FUNCTION_BLOCK FB_SimuMoverAxis
VAR_INPUT
    xIN_StopMover : BOOL; // stop the mover from movinf
END_VAR
VAR_OUTPUT
    outSimuCurrentPos : Pos2D_t; // Mover position, expressed as slot number
    outSimuCurrentRot : INT;     // mover current rotation
    isInPos           : BOOL;    // true when targetPos = currentPos
END_VAR
VAR
    // with tick rate at 10ms, a value of 10 gives us 1m/s
    _Velocity    : LREAL := 0;     // Mover velocity, expressed as mm per tick, max is 10m/s
    _ErrorState  : INT   := 0;     // error state, not used
    _TargetPos   : LREAL := 0;     // last target pos
    _CurrentPos  : LREAL := 0;     // Current Pos, but with more resolution than the pixel
    _IsColliding : BOOL  := FALSE; // When true, the mover should not move
    _LastPos     : LREAL := 0;     // last position, used to trigger the xStuck flag
    _xStuck      : BOOL;           // true when the axis does not move
    _willCollide : BOOL := FALSE;  // TRUE if a collision will occure with the current velocity

    {attribute 'hide'}
    _lrNextStopPos : LREAL; // local variable used to get next stop

    _iID : INT := 0; // instance ID, is set during FB_Init using the value of _iInstanceCounter 
	
	_CurrentDir : MoverDirection_e := MoverDirection_e.Farward;
END_VAR

VAR_TEMP
	_MoverAccel : LREAL;	// Mover acceleration, can be positive or negative depending on the direction
END_VAR

VAR CONSTANT
    MAX_POS            : LREAL := CONST.MAX_TRACK_LENGTH; // should be defined elsewhere ...
    MAX_SIZE           : LREAL := CONST.MAX_MOVER_SIZE;   // Maxium size of the mover
    //MOVER_ACCEL        : LREAL := 0.1;                      // Mover acceleration, in mm/tick^2
    //MOVER_VELOCITY_MAX : LREAL := 20;                     // Mover velocity, expressed as mm per tick, max is 10m/s
    MOVER_VELOCITY_MIN : LREAL := 1;                      // Mover velocity, expressed as mm per tick, max is 10m/s
END_VAR
VAR_STAT
    _iInstanceCounter : INT := 1; // instance counter
END_VAR

IF NOT xIN_StopMover THEN // Do not change momemtum when we stop the movers from HMI
    IF MoverDirection_e.Farward = THIS^._CurrentDir THEN
        _MoverAccel := SIMU.lrAccelMover;
    ELSE
        _MoverAccel := -SIMU.lrAccelMover;
    END_IF

    IF NOT _IsColliding THEN

        IF THIS^.GetStopLen(_Velocity, SIMU.lrAccelMover) >= DistToTravel(_CurrentPos, _TargetPos) OR
           THIS^._willCollide THEN
            _Velocity := _Velocity - _MoverAccel;

        ELSIF SIMU.lrSpeedMover > ABS(_Velocity) AND _CurrentPos <> _TargetPos THEN
            _Velocity := _Velocity + _MoverAccel;

        END_IF
    ELSE
        _Velocity := _Velocity - _MoverAccel;
    END_IF
END_IF

// protect max and min speed
IF SIMU.lrSpeedMover < ABS(_Velocity) THEN
    IF MoverDirection_e.Farward = THIS^._CurrentDir THEN
        _Velocity := SIMU.lrSpeedMover;
    ELSE
        _Velocity := -SIMU.lrSpeedMover;
    END_IF
ELSIF ABS(_Velocity) < MOVER_VELOCITY_MIN THEN
    IF MoverDirection_e.Farward = THIS^._CurrentDir THEN
        _Velocity := MOVER_VELOCITY_MIN;
    ELSE
        _Velocity := -MOVER_VELOCITY_MIN;
    END_IF
END_IF

IF NOT _IsColliding AND NOT xIN_StopMover THEN

    IF DistToTravel(_CurrentPos, _TargetPos) > ABS(_Velocity) THEN
        _CurrentPos := _CurrentPos + _Velocity;

    ELSE
        _CurrentPos := _TargetPos;
        _Velocity   := 0;

    END_IF
END_IF

IF _CurrentPos >= MAX_POS THEN
    _CurrentPos := _CurrentPos - MAX_POS;
    // we prevent the stuck flag to be true at the end of the track
    THIS^._LastPos := THIS^._LastPos - MAX_POS;
END_IF

isInPos := EqualDelta(_CurrentPos, _TargetPos, 1.0); // we use delta comparison beacause axis is always at a low value 
outSimuCurrentPos
    := THIS^.ResolvePos(this^.CurrentPos, outSimuCurrentRot);

_xStuck        := (THIS^._CurrentPos < (THIS^._LastPos + _Velocity)) AND NOT isInPos;
THIS^._LastPos := THIS^._CurrentPos;

PROPERTY CurrentPos : LREAL
GET
IF CONST.USE_SIMULATION THEN
    CurrentPos := _CurrentPos;
ELSE
    CurrentPos := TO_LREAL(gMoverAxis.I_BuR_MoverAxis.asStruct[THIS^._iID].diCurrentPos_um) / 1000.0;
END_IF
END_GET
SET
END_SET
END_PROPERTY

PROPERTY CurrentVelocity : LREAL
GET
CurrentVelocity := THIS^._Velocity;
END_GET
SET
END_SET
END_PROPERTY

METHOD FB_init : BOOL
VAR_INPUT
    bInitRetains : BOOL; // if TRUE, the retain variables are initialized (warm start / cold start)
    bInCopyCode  : BOOL; // if TRUE, the instance afterwards gets moved into the copy code (online change)

    PosInit : LREAL; // initial position at startup
END_VAR
THIS^._iID := THIS^._iInstanceCounter;
THIS^._iInstanceCounter := THIS^._iInstanceCounter +1;
IF PosInit < THIS^.MAX_POS THEN
    THIS^._CurrentPos := PosInit;
ELSE
    THIS^._CurrentPos := 0;
END_IF
END_METHOD

METHOD PRIVATE GetStopLen : LREAL
VAR_INPUT
    currentVelocity : LREAL;
    currentAccel    : LREAL;
END_VAR
VAR
    tickToStop : INT;
END_VAR
// This function search the position we will get if we stop now
//
// (velocity)
//     ^          _________   <- we are here, at the end of the top slope
//     |        /          \
//     |       /            \
//     |   ___/              \______
//     |     
//     ┼------------------------------>  (time)
//
// (position)
//     ^ 
//     |                      _________
//     |                  .../
//     |               ../    ^
//     |            ../       |
//     |          ../         we search this position
//     |   ___.../
//     | 
//     ┼------------------------------>  (time)

IF currentAccel <= 0 THEN
    ASSERT(currentAccel > 0);
    RETURN;
END_IF

// TO_INT floor the result, and we need at least 1 tick to stop
tickToStop := TO_INT(currentVelocity / currentAccel) + 1;

GetStopLen := tickToStop * currentVelocity / 2;
END_METHOD

// only check the collision in one way, this prevent
// all the mover chain to be stucked
METHOD IsColliding : BOOL
VAR_INPUT
    nextMover : REFERENCE TO FB_SimuMoverAxis;
END_VAR
IsColliding := FALSE;

IF DistToTravel(THIS^.CurrentPos, nextMover.CurrentPos) <= CONST.MAX_MOVER_SIZE THEN
    IsColliding := TRUE;

END_IF

THIS^._IsColliding := IsColliding;
END_METHOD

METHOD PUBLIC MoveTo : REFERENCE TO FB_SimuMoverAxis
VAR_INPUT
    Position : LREAL; // move the axis to this position
END_VAR
THIS^._TargetPos := Position;
THIS^._CurrentDir := MoverDirection_e.Farward;
isInPos := THIS^._CurrentPos = THIS^._TargetPos;
MoveTo REF= THIS^;
END_METHOD

// Move relatively of this position
// With this function, a negative value move the mover at the reverse direction
METHOD RelMoveTo : REFERENCE TO FB_SimuMoverAxis
VAR_INPUT
    RelativePos : LREAL; // move the axis to this amount¨
END_VAR
THIS^._TargetPos := THIS^._TargetPos + RelativePos;

IF RelativePos >= 0 THEN
    THIS^._CurrentDir := MoverDirection_e.Farward;
ELSE
    THIS^._CurrentDir := MoverDirection_e.Reverse;
END_IF

isInPos   := THIS^._CurrentPos = THIS^._TargetPos;
RelMoveTo REF= THIS^;
END_METHOD

METHOD ResolvePos : Pos2D_t
VAR_INPUT
    inX      : LREAL;
    rotation : REFERENCE TO INT;
END_VAR
VAR CONSTANT
    (* The track has this dimension in reality
              __________
     1000mm (___________) 1000 mm
              4000 mm
			  
     and we map it like that:
	   __   80 (radius)
	  |  |
	  |  |  800
	  |  |
	  |__|
	        80 (raidus)
    *)
    START_X     : DINT  := 0;
    START_Y     : DINT  := 0;
    MAX_SIMU_DX : DINT  := 120;
    MAX_SIMU_DY : DINT  := 800;
    RADIUS_X    : LREAL := 60.0;
    RADIUS_Y    : LREAL := 80.0;

    FIRST_RADIUS_START  : LREAL := 4000;
    FIRST_RADIUS_END    : LREAL := 5000;
    SECOND_RADIUS_START : LREAL := 9000;
    SECOND_RADIUS_END   : LREAL := 10000;
END_VAR

VAR
    x_rad_calc : LREAL;
    y_rad_calc : LREAL;
    FACTOR_Y   : LREAL;
END_VAR
FACTOR_Y := FIRST_RADIUS_START / MAX_SIMU_DY;

IF inX < 0 THEN
    ResolvePos.x := START_X;
    ResolvePos.y := START_Y;
    rotation     := 0;

ELSIF inX >= 0 AND inX <= FIRST_RADIUS_START THEN
    ResolvePos.x := START_X;
    ResolvePos.y := START_Y + TO_DINT(inX / FACTOR_Y);
    rotation     := 0;

ELSIF inX > FIRST_RADIUS_START AND inX < FIRST_RADIUS_END THEN

    // should go between -1RAD and +1RAD
    x_rad_calc   := ((inX - FIRST_RADIUS_START) * 2 / (FIRST_RADIUS_END - FIRST_RADIUS_START) - 1) * PI / 2;
    ResolvePos.x := TO_DINT(SIN(x_rad_calc) * RADIUS_X) + START_X + TO_DINT(RADIUS_X);

    // should go from 0RAD to 1RAD, then 0RAD
    y_rad_calc   := (1 - (inX - FIRST_RADIUS_START) * 2 / (FIRST_RADIUS_END - FIRST_RADIUS_START)) * PI / 2;
    ResolvePos.y := TO_DINT(COS(y_rad_calc) * RADIUS_Y + START_Y + MAX_SIMU_DY);

    rotation := TO_INT(SIN(x_rad_calc) * 90 + 90);

ELSIF inX >= FIRST_RADIUS_END AND inX <= SECOND_RADIUS_START THEN
    ResolvePos.x := START_X + MAX_SIMU_DX;
    ResolvePos.y := START_Y + MAX_SIMU_DY - TO_DINT((inX - FIRST_RADIUS_END) / FACTOR_Y);
    rotation     := 180;

ELSIF inX > SECOND_RADIUS_START AND inX < SECOND_RADIUS_END THEN
    // should go between -1RAD and +1RAD
    x_rad_calc   := ((inX - SECOND_RADIUS_START) * 2 / (SECOND_RADIUS_END - SECOND_RADIUS_START) - 1) * PI / 2;
    ResolvePos.x := START_X - TO_DINT(SIN(x_rad_calc) * RADIUS_X) + TO_DINT(RADIUS_X);

    // should go from 0RAD to 1RAD, then 0RAD
    y_rad_calc   := (1 - (inX - SECOND_RADIUS_START) * 2 / (SECOND_RADIUS_END - SECOND_RADIUS_START)) * PI / 2;
    ResolvePos.y := START_Y - TO_DINT(COS(y_rad_calc) * RADIUS_Y);

    rotation := TO_INT(SIN(x_rad_calc) * 90 + 270);

ELSE
    ResolvePos.x := START_X;
    ResolvePos.y := START_Y;
    rotation     := 0;

END_IF
END_METHOD

METHOD ToString : STRING
VAR_INPUT
END_VAR
VAR
END_VAR
ToString := CONCAT('FB_SimuMoverAxis_', TO_STRING(THIS^._iID));
END_METHOD

// Use this method in a collider manager so the simu axis 
// will know when to stop itself
METHOD WillCollide : BOOL
VAR_INPUT
    nextMover : REFERENCE TO FB_SimuMoverAxis;
END_VAR
VAR
    diffVelocity : LREAL;
END_VAR
THIS^._willCollide := FALSE;
diffVelocity       := 0;

// If the 2 movers are moving tarwards each other
IF (THIS^._Velocity > 0) AND (nextMover.CurrentVelocity < 0) THEN
    diffVelocity := SQRT(THIS^._Velocity * THIS^._Velocity + (nextMover.CurrentVelocity * nextMover.CurrentVelocity));

    // If the 2 movers are moving in the same direction
ELSE
    IF ABS(THIS^._Velocity) > ABS(nextMover.CurrentVelocity) THEN
        diffVelocity :=
            SQRT(THIS^._Velocity * THIS^._Velocity - (nextMover.CurrentVelocity * nextMover.CurrentVelocity));
    END_IF
END_IF

THIS^._willCollide
    := DistToTravel(THIS^.CurrentPos, nextMover.CurrentPos) <=
       THIS^.GetStopLen(diffVelocity, SIMU.lrAccelMover) + CONST.MAX_MOVER_SIZE;

WillCollide := THIS^._willCollide;
END_METHOD

PROPERTY xStuck : BOOL
GET
xStuck := _xStuck;
END_GET
SET
END_SET
END_PROPERTY

END_FUNCTION_BLOCK

(* stored: Version 1.1.0.1, ProductVersion 3.1.4024.6
   POU FB_SimuMoverAxis: Id {017f40e2-f1f1-4976-849d-fa06ef0a4cb5}, SpecialFunc None
   Property CurrentPos: Id {c358a281-78eb-40b2-b89a-a18eff26d260}
   Get Get: Id {b61bd9b1-08af-4926-b858-85c8eb24b2db}
   Set Set: Id {c5f537f5-5d8c-45ad-a5c5-df77003f95bc}
   Property CurrentVelocity: Id {b8df0f34-d17e-487c-9bfd-ce3e7601077b}
   Get Get: Id {4eba8587-6625-4315-9a97-80fc827c5652}
   Set Set: Id {93f7958f-bf31-42ad-9468-d8476b3f9641}
   Method FB_init: Id {b65ea979-747b-41ba-bf6e-1edaa259930c}
   Method GetStopLen: Id {b13fe67a-491d-4b80-98f9-d811ecbf3cca}
   Method IsColliding: Id {57cc6fd2-d942-4280-a88c-6e6aadeff802}
   Method MoveTo: Id {27ffc6e2-2e43-4eb2-aced-4a958cfe10ec}
   Method RelMoveTo: Id {63f20b0f-13f1-4d11-9d44-19187e776860}
   Method ResolvePos: Id {16435a25-f091-4756-88c1-e63202a0b39c}
   Method ToString: Id {76b4f3b8-9490-4f7f-bb39-de0a0d71ce03}
   Method WillCollide: Id {0d97bec0-b7d4-4420-83e5-72f1aaaf45d7}
   Property xStuck: Id {f828bdb7-715a-4f3c-9d48-98ebe68f4f98}
   Get Get: Id {9f868acf-4f41-4320-ace9-846357c4a7b6}
   Set Set: Id {717d36c5-f749-4432-8cb5-c2f33a7a865e} *)
